{attribute 'qualified_only'}
VAR_GLOBAL CONSTANT
  NUM_EVENTS: INT := 4;
  NUM_EVENT_HISTORY: INT := 10;
  NUM_CONCURRENT_ALARMS: INT := 10;
  NUM_LOGGER: INT := 5;
END_VAR

(* stored: Version 1.1.0.1, ProductVersion 3.1.4024.9
   GVL Properties: Id {f4d96ff7-2767-4dda-aedb-114ebae1033c}, ParameterList True *)
